(* PLC project Unnamed, Unknown Unnamed 1 *)
(* stored: creationDateTime 2023-03-10T10:37:17, modificationDateTime 2023-03-15T15:56:42 *)

(* https://www.gds2.de/fileadmin/umwelttechnik/umwelttechnik/skripte/steuerungstechnik_ut_2017.pdf, 2.12 *)
FUNCTION_BLOCK Thermometer_Code_System
  VAR_INPUT
    IN1 : BOOL;
    IN2 : BOOL;
    IN3 : BOOL;
    IN4 : BOOL;
  END_VAR
  VAR_OUTPUT
    OUT1 : BOOL;
    OUT2 : BOOL;
    OUT3 : BOOL;
  END_VAR
  VAR  (* added by the conversion: wires and edge detectors of the diagram *)
    _AND26_OUT : BOOL;
  END_VAR

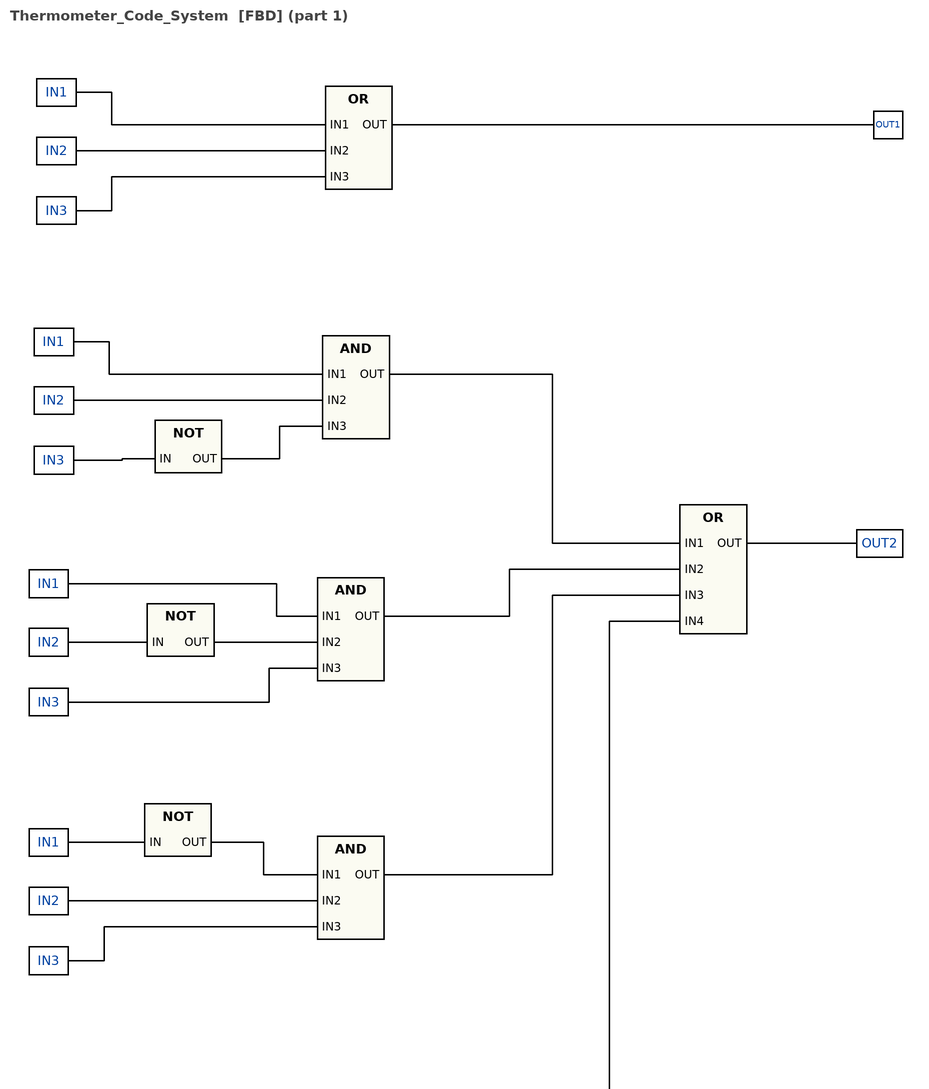
(* FBD diagram, written out as Structured Text *)
OUT1 := IN1 OR IN2 OR IN3;
_AND26_OUT := IN1 AND IN2 AND IN3;
OUT2 := IN1 AND IN2 AND NOT IN3 OR IN1 AND NOT IN2 AND IN3 OR NOT IN1 AND IN2 AND IN3 OR _AND26_OUT;
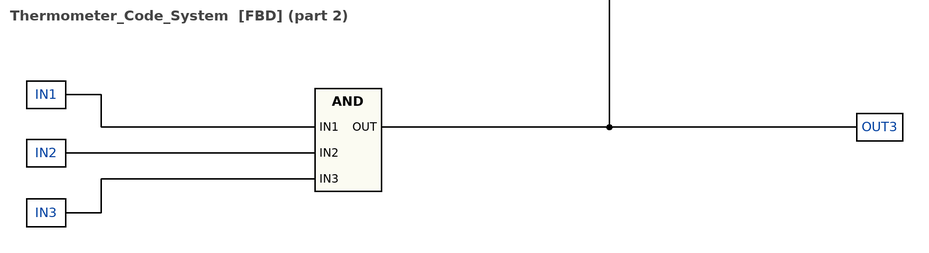
OUT3 := _AND26_OUT;
END_FUNCTION_BLOCK

CONFIGURATION config
  RESOURCE resource1 ON PLC
  END_RESOURCE
END_CONFIGURATION
